TYPE Frame :
STRUCT
	Name : STRING;
	X : REAL;
	Y : REAL;
END_STRUCT
END_TYPE

(* stored: Version 1.1.0.1, ProductVersion 3.1.4024.9
   DUT Frame: Id {1b792bef-e222-4263-bf55-2d37b3f66bbf} *)
